// Converts a T_Size value to a DINT value.
FUNCTION F_SizeToDint : DINT // The converted DINT value from the given T_Size.
VAR_INPUT
	Size : T_Size; // The input size to be converted.
END_VAR

F_SizeToDint := TO_DINT(LIMIT(0, Size, TO_UDINT(GVL_TypeValueLimits.DINT_MAX)));

END_FUNCTION

(* stored: Version 1.1.0.1
   POU F_SizeToDint: Id {7e77e26b-3566-0862-28eb-e27f37aed3cf}, SpecialFunc None *)
